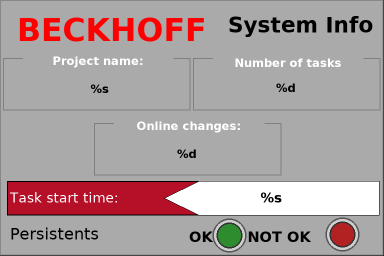
VISUALIZATION PH_SystemInfo  // 384x256
    Rectangle (0,0 384x256)
    Label (9,10 206x40), "BECKHOFF"
    Label (217,10 168x30), "System Info"
    RoundedRectangle (3,58 187x52)
    Rectangle (23,46 150x30), "Project name:"
    RoundedRectangle (193,58 187x52)
    Rectangle (213,48 150x30), "Number of tasks"
    RoundedRectangle (7,181 205x34), "Task start time:"
    Polygon (164,198) (199,181) (379,181) (379,215) (199,215), "%s", text variable: P_SystemInfo.sStartTime
    RoundedRectangle (94,123 187x52)
    Rectangle (114,111 150x30), "Online changes:"
    Label (7,219 251x30), "Persistents"
    Lamp1 (323,215 39x39), variable: P_SystemInfo.bError, style: Lamp-Lamp1-Red
    Rectangle (25,74 150x30), "%s", text variable: P_SystemInfo.sProjectName
    Rectangle (211,73 150x30), "%d", text variable: P_SystemInfo.nTaskCount
    Rectangle (112,139 150x30), "%d", text variable: P_SystemInfo.nOnlineChangesCOunt
    Lamp1 (210,216 39x39), variable: P_SystemInfo.bOK, style: Lamp-Lamp1-Green
    Label (145,222 210x30), "OK NOT OK"
END_VISUALIZATION

(* stored: Version 1.1.0.1, ProductVersion 3.1.4024.5
   Visu PH_SystemInfo: Id {bab3a2b3-6dcc-46ac-a370-51de0314ebb0} *)
